ADAPTER PICKER_STATE_BA (* Adapter Interface for Model -> View *)
  (* Standard: 61499-1 *)
  (* Version 0.2, 2003-12-05, JHC, Rockwell Automation, Changed name from NEWADAPTER *)
  (* Version 0.1, 2002-01-08, JHC, Rockwell Automation, Added IND/RSP, renamed data, added sequences. *)
  (* Version 0.0, 2000-05-27, JHC, Rockwell Automation *)
  (* Compiler header: package fb.rt.pnp; *)
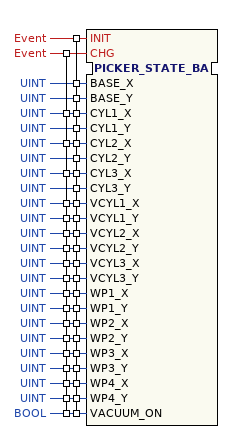
  EVENT_INPUT
    INIT WITH BASE_X, BASE_Y, CYL1_Y, CYL2_Y, CYL1_X, CYL2_X, VCYL1_X, VCYL1_Y, WP1_X, WP1_Y, VACUUM_ON, WP2_X, WP2_Y, WP3_X, WP3_Y, CYL3_X, CYL3_Y, VCYL2_X, VCYL2_Y, VCYL3_X, VCYL3_Y, WP4_X, WP4_Y;
    CHG WITH CYL1_X, CYL2_X, VCYL1_X, VCYL1_Y, WP1_X, WP1_Y, VACUUM_ON, WP2_X, WP2_Y, WP3_X, WP3_Y, VCYL2_X, VCYL2_Y, VCYL3_X, VCYL3_Y, WP4_X, WP4_Y, CYL3_X; (* Change of state *)
  END_EVENT
  VAR_INPUT
    BASE_X : UINT; (* Request Data from Socket *)
    BASE_Y : UINT; (* Request Data from Socket *)
    CYL1_X : UINT; (* Request Data from Socket *)
    CYL1_Y : UINT; (* Request Data from Socket *)
    CYL2_X : UINT; (* Response Data from Socket *)
    CYL2_Y : UINT; (* Request Data from Socket *)
    CYL3_X : UINT; (* Response Data from Socket *)
    CYL3_Y : UINT; (* Request Data from Socket *)
    VCYL1_X : UINT; (* Response Data from Socket *)
    VCYL1_Y : UINT; (* Response Data from Socket *)
    VCYL2_X : UINT; (* Response Data from Socket *)
    VCYL2_Y : UINT; (* Response Data from Socket *)
    VCYL3_X : UINT; (* Response Data from Socket *)
    VCYL3_Y : UINT; (* Response Data from Socket *)
    WP1_X : UINT; (* Response Data from Socket *)
    WP1_Y : UINT; (* Response Data from Socket *)
    WP2_X : UINT;
    WP2_Y : UINT;
    WP3_X : UINT;
    WP3_Y : UINT;
    WP4_X : UINT;
    WP4_Y : UINT;
    VACUUM_ON : BOOL; (* Response Data from Socket *)
  END_VAR
  SERVICE SOCKET/PLUG
    SEQUENCE request_confirm
      SOCKET.REQ(REQD) -> PLUG.REQ(REQD);
      PLUG.CNF(CNFD) -> SOCKET.CNF(CNFD);
    END_SEQUENCE
    SEQUENCE indication_response
      PLUG.IND(INDD) -> SOCKET.IND(INDD);
      SOCKET.RSP(RSPD) -> PLUG.RSP(RSPD);
    END_SEQUENCE
  END_SERVICE
END_ADAPTER
